(* CODESYS project GVL_MACHINE.gvl.xml

Project tree, tasks and I/O mapping:
  global variables GVL_MACHINE
*)

// GVL_MACHINE
{attribute 'qualified_only'}
VAR_GLOBAL
	Command : ARRAY [1..3] OF ST_MACHINE_COMMAND; // Команды станков и робота
	Status  : ARRAY [1..3] OF ST_MACHINE_PUBLIC; // Рабочие статусы станков
	Diag    : ARRAY [1..3] OF ST_MACHINE_DIAG; // Состояния автоматов станков
	Error   : ARRAY [1..3] OF ST_MACHINE_ERRORS; // Ошибки станков
END_VAR
